INTERFACE I_LinkFactory

METHOD PUBLIC Create : I_Link
VAR_INPUT
	LinkId : T_MAXSTRING;
	LinkSourceNode : I_Node;
	LinkSourcePortName : STRING;
	LinkDestinationNode : I_Node;
	LinkDestinationPortName : STRING;
END_VAR
END_METHOD

END_INTERFACE

(* stored: Version 1.1.0.1, ProductVersion 3.1.4024.12
   Itf I_LinkFactory: Id {658e30ce-4938-083c-272d-50ec4dc45dfa}
   Method Create: Id {0fc03fb6-f4de-0601-0233-3c97068405c8} *)
